PROGRAM RS485_prg
VAR
	COM_485 : FB_485;
	COMportControl_MASTER: SerialLineControl;
	COMportControlError_MASTER : BOOL;
	COMportControlErrorID_MASTER : ComError_t;	

END_VAR


COM_485.update();

COMportControl_MASTER(
	Mode:=SERIALLINEMODE_EL6_22B,
	pComIn:= ADR(GVL.COMin_EL6021_MASTER),
	pComOut:= ADR(GVL.COMout_EL6021_MASTER),
	SizeComIn:= UINT_TO_INT(SIZEOF(GVL.COMin_EL6021_MASTER)),
	TxBuffer:= GVL.TxBuffer_MASTER,
	RxBuffer:=GVL.RxBuffer_MASTER,
	Error => COMportControlError_MASTER,
	ErrorID => COMportControlErrorID_MASTER);

END_PROGRAM

(* stored: Version 1.1.0.1, ProductVersion 3.1.4024.15
   POU RS485_prg: Id {f7892673-7b64-41e0-b2f7-55c10529511e}, SpecialFunc None *)
